% RSLogix 500 project P10 - Pump Protection.RSS, saved by version 8.30.00.16 %
PROJECT "P10"    % processor: Bul.1763 MicroLogix 1100 Series B %

PROGRAM FILES
  LAD 2 "MAIN"  3 rungs
  LAD 3 "I/O"  7 rungs
  LAD 4 "PRC. LOGIC"  16 rungs

DATA FILES
  O0 OUTPUT  4 elements
  I1 INPUT  6 elements
  S2 STATUS  66 elements
  B3 BINARY  2 elements
  T4 TIMER  3 elements
  C5 COUNTER  1 elements
  R6 CONTROL  1 elements
  N7 INTEGER  6 elements
  F8 FLOAT  1 elements

LADDER 2 "MAIN"
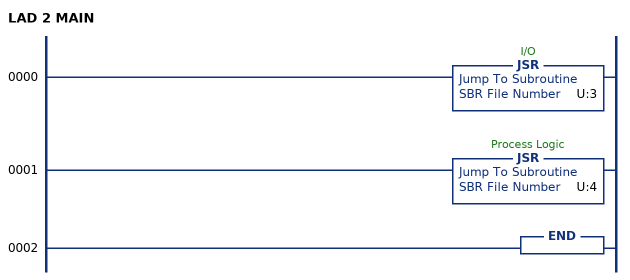
% Rung: 0 %
SOR JSR U:3 EOR
%   U:3  "I/O" %
% Rung: 1 %
SOR JSR U:4 EOR
%   U:4  "Process Logic" %
% Rung: 2 %
SOR END EOR

LADDER 3 "I/O"
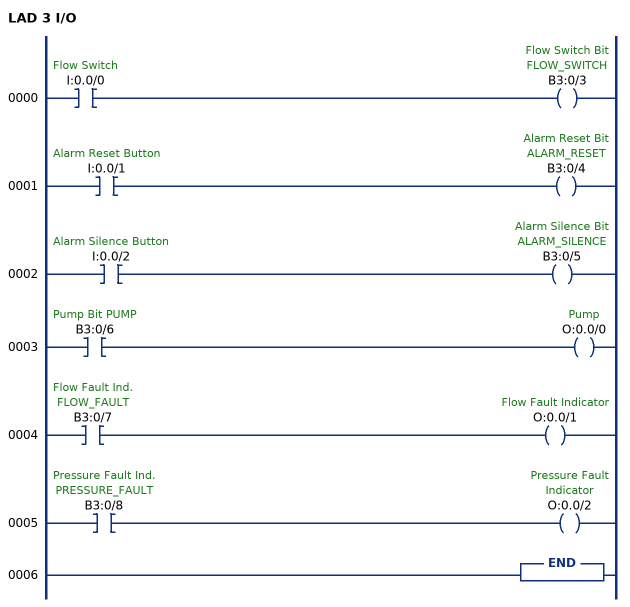
% Rung: 0 %
SOR XIC I:0.0/0 OTE B3:0/3 EOR
%   I:0.0/0  "Flow Switch" %
%   B3:0/3  FLOW_SWITCH  "Flow Switch Bit" %
% Rung: 1 %
SOR XIC I:0.0/1 OTE B3:0/4 EOR
%   I:0.0/1  "Alarm Reset Button" %
%   B3:0/4  ALARM_RESET  "Alarm Reset Bit" %
% Rung: 2 %
SOR XIC I:0.0/2 OTE B3:0/5 EOR
%   I:0.0/2  "Alarm Silence Button" %
%   B3:0/5  ALARM_SILENCE  "Alarm Silence Bit" %
% Rung: 3 %
SOR XIC B3:0/6 OTE O:0.0/0 EOR
%   B3:0/6  PUMP  "Pump Bit" %
%   O:0.0/0  "Pump" %
% Rung: 4 %
SOR XIC B3:0/7 OTE O:0.0/1 EOR
%   B3:0/7  FLOW_FAULT  "Flow Fault Ind." %
%   O:0.0/1  "Flow Fault Indicator" %
% Rung: 5 %
SOR XIC B3:0/8 OTE O:0.0/2 EOR
%   B3:0/8  PRESSURE_FAULT  "Pressure Fault Ind." %
%   O:0.0/2  "Pressure Fault Indicator" %
% Rung: 6 %
SOR END EOR

LADDER 4 "PRC. LOGIC"
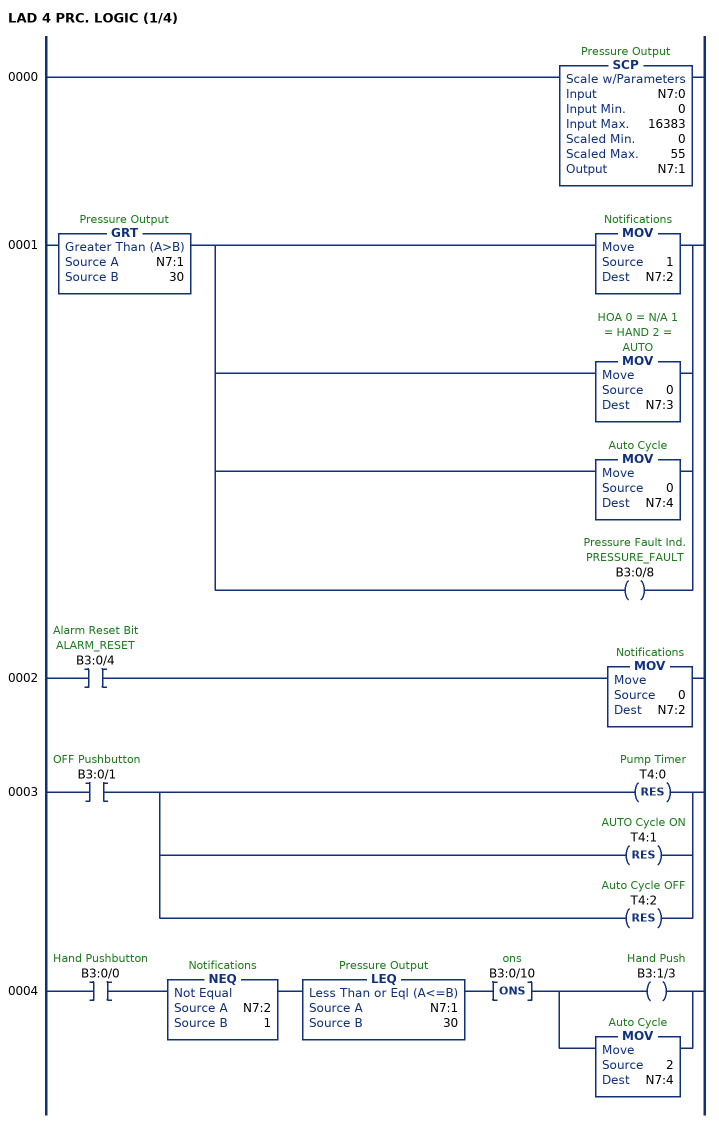
% Rung: 0 %
SOR SCP N7:0 0 16383 0 55 N7:1 EOR
%   N7:0  "Pressure Sensor" %
%   N7:1  "Pressure Output" %
% Rung: 1 %
SOR GRT N7:1 30 BST MOV 1 N7:2 NXB MOV 0 N7:3 NXB MOV 0 N7:4 NXB OTE B3:0/8 BND EOR
%   N7:1  "Pressure Output" %
%   N7:2  "Notifications" %
%   N7:3  "HOA 0 = N/A 1 = HAND 2 = AUTO" %
%   N7:4  "Auto Cycle" %
%   B3:0/8  PRESSURE_FAULT  "Pressure Fault Ind." %
% Rung: 2 %
SOR XIC B3:0/4 MOV 0 N7:2 EOR
%   B3:0/4  ALARM_RESET  "Alarm Reset Bit" %
%   N7:2  "Notifications" %
% Rung: 3 %
SOR XIC B3:0/1 BST RES T4:0 NXB RES T4:1 NXB RES T4:2 BND EOR
%   B3:0/1  "OFF Pushbutton" %
%   T4:0  "Pump Timer" %
%   T4:1  "AUTO Cycle ON" %
%   T4:2  "Auto Cycle OFF" %
% Rung: 4 %
SOR XIC B3:0/0 NEQ N7:2 1 LEQ N7:1 30 ONS B3:0/10 BST OTE B3:1/3 NXB MOV 2 N7:4 BND EOR
%   B3:0/0  "Hand Pushbutton" %
%   N7:2  "Notifications" %
%   N7:1  "Pressure Output" %
%   B3:0/10  "ons" %
%   B3:1/3  "Hand Push" %
%   N7:4  "Auto Cycle" %

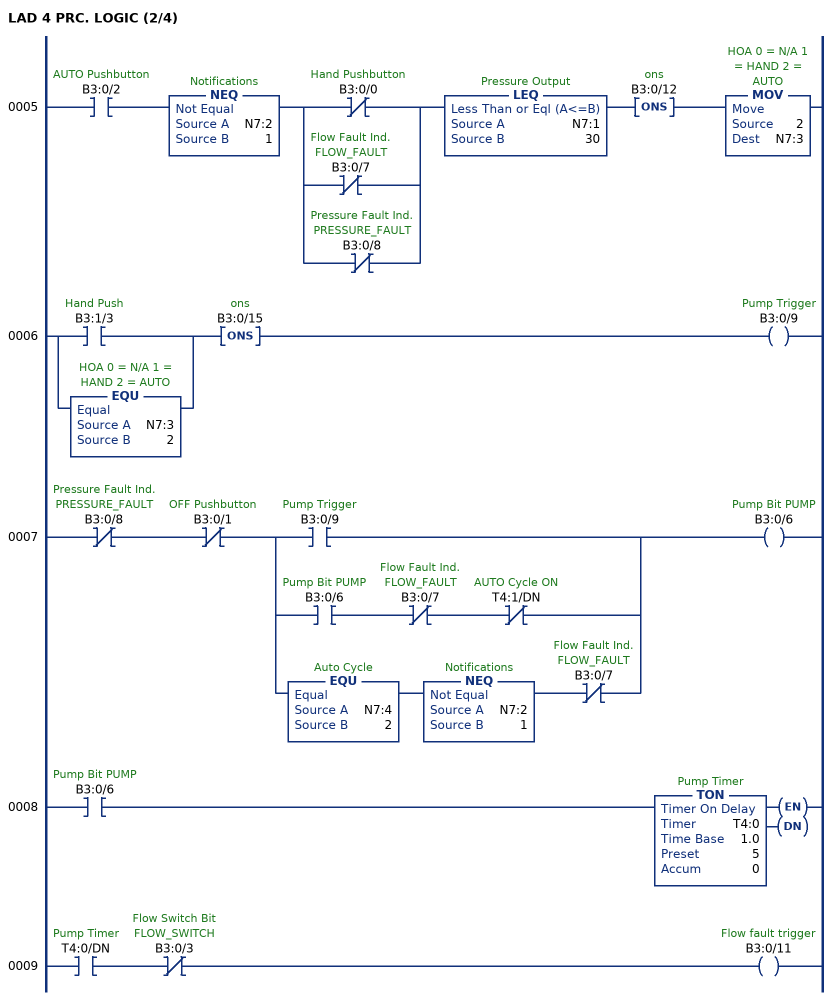
% Rung: 5 %
SOR XIC B3:0/2 NEQ N7:2 1 BST XIO B3:0/0 NXB XIO B3:0/7 NXB XIO B3:0/8 BND LEQ N7:1 30 ONS B3:0/12 MOV 2 N7:3 EOR
%   B3:0/2  "AUTO Pushbutton" %
%   N7:2  "Notifications" %
%   B3:0/0  "Hand Pushbutton" %
%   B3:0/7  FLOW_FAULT  "Flow Fault Ind." %
%   B3:0/8  PRESSURE_FAULT  "Pressure Fault Ind." %
%   N7:1  "Pressure Output" %
%   B3:0/12  "ons" %
%   N7:3  "HOA 0 = N/A 1 = HAND 2 = AUTO" %
% Rung: 6 %
SOR BST XIC B3:1/3 NXB EQU N7:3 2 BND ONS B3:0/15 OTE B3:0/9 EOR
%   B3:1/3  "Hand Push" %
%   N7:3  "HOA 0 = N/A 1 = HAND 2 = AUTO" %
%   B3:0/15  "ons" %
%   B3:0/9  "Pump Trigger" %
% Rung: 7 %
SOR XIO B3:0/8 XIO B3:0/1 BST XIC B3:0/9 NXB XIC B3:0/6 XIO B3:0/7 XIO T4:1/DN NXB EQU N7:4 2 NEQ N7:2 1 XIO B3:0/7 BND OTE B3:0/6 EOR
%   B3:0/8  PRESSURE_FAULT  "Pressure Fault Ind." %
%   B3:0/1  "OFF Pushbutton" %
%   B3:0/9  "Pump Trigger" %
%   B3:0/6  PUMP  "Pump Bit" %
%   B3:0/7  FLOW_FAULT  "Flow Fault Ind." %
%   T4:1  "AUTO Cycle ON" %
%   N7:4  "Auto Cycle" %
%   N7:2  "Notifications" %
% Rung: 8 %
SOR XIC B3:0/6 TON T4:0 1.0 5 0 EOR
%   B3:0/6  PUMP  "Pump Bit" %
%   T4:0  "Pump Timer" %
% Rung: 9 %
SOR XIC T4:0/DN XIO B3:0/3 OTE B3:0/11 EOR
%   T4:0  "Pump Timer" %
%   B3:0/3  FLOW_SWITCH  "Flow Switch Bit" %
%   B3:0/11  "Flow fault trigger" %

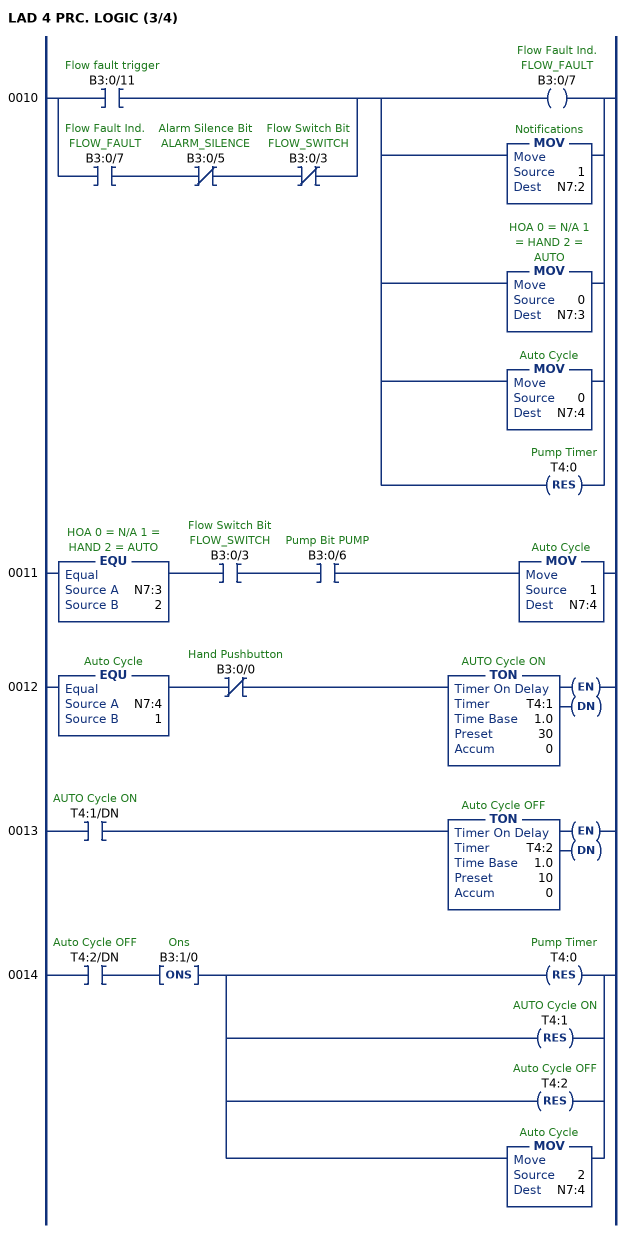
% Rung: 10 %
SOR BST XIC B3:0/11 NXB XIC B3:0/7 XIO B3:0/5 XIO B3:0/3 BND BST OTE B3:0/7 NXB MOV 1 N7:2 NXB MOV 0 N7:3 NXB MOV 0 N7:4 NXB RES T4:0 BND EOR
%   B3:0/11  "Flow fault trigger" %
%   B3:0/7  FLOW_FAULT  "Flow Fault Ind." %
%   B3:0/5  ALARM_SILENCE  "Alarm Silence Bit" %
%   B3:0/3  FLOW_SWITCH  "Flow Switch Bit" %
%   N7:2  "Notifications" %
%   N7:3  "HOA 0 = N/A 1 = HAND 2 = AUTO" %
%   N7:4  "Auto Cycle" %
%   T4:0  "Pump Timer" %
% Rung: 11 %
SOR EQU N7:3 2 XIC B3:0/3 XIC B3:0/6 MOV 1 N7:4 EOR
%   N7:3  "HOA 0 = N/A 1 = HAND 2 = AUTO" %
%   B3:0/3  FLOW_SWITCH  "Flow Switch Bit" %
%   B3:0/6  PUMP  "Pump Bit" %
%   N7:4  "Auto Cycle" %
% Rung: 12 %
SOR EQU N7:4 1 XIO B3:0/0 TON T4:1 1.0 30 0 EOR
%   N7:4  "Auto Cycle" %
%   B3:0/0  "Hand Pushbutton" %
%   T4:1  "AUTO Cycle ON" %
% Rung: 13 %
SOR XIC T4:1/DN TON T4:2 1.0 10 0 EOR
%   T4:1  "AUTO Cycle ON" %
%   T4:2  "Auto Cycle OFF" %
% Rung: 14 %
SOR XIC T4:2/DN ONS B3:1/0 BST RES T4:0 NXB RES T4:1 NXB RES T4:2 NXB MOV 2 N7:4 BND EOR
%   T4:2  "Auto Cycle OFF" %
%   B3:1/0  "Ons" %
%   T4:0  "Pump Timer" %
%   T4:1  "AUTO Cycle ON" %
%   N7:4  "Auto Cycle" %

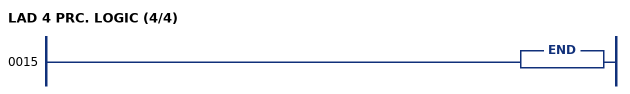
% Rung: 15 %
SOR END EOR

OTHER DOCUMENTED ADDRESSES
  B3:0/13  "ons"
  B3:0/14  "Hand.pump trigger"
  B3:1/4  "ons"
  N7:5  "Pump ON/OFF"

DATA TABLE (non-zero values as saved)
DATA T4
% .PRE .ACC %
% T4:0 % 5 0
% T4:1 % 30 0
% T4:2 % 10 0
